TYPE ST_LogEntry :
STRUCT
    sMessage : STRING(255);
    dtTimestamp : DATE_AND_TIME;
    eType : E_LogType;
	sTypeName : STRING(20);
END_STRUCT
END_TYPE

(* stored: Version 1.1.0.1
   DUT ST_LogEntry: Id {2a7b43e3-1021-4bad-901e-295452d5e9d1} *)
